{attribute 'linkalways'} 
{attribute 'no_explicit_call' := 'This FB is a CLASS and must be accessed using methods or properties'}
{attribute 'enable_dynamic_creation'}
FUNCTION_BLOCK Node_F_VN_ConvexHullPointsExp EXTENDS VisionNode
VAR
    ipPointSet : _ITcVnContainer;
    ipConvexHull : _ITcVnContainer;
    bClockwise : _BOOL(FALSE);
    hrPrev : _HRESULT(S_OK);
	hresult : _HRESULT(S_OK);
END_VAR

METHOD PUBLIC  Clone : I_Node
VAR
	pNode : POINTER TO Node_F_VN_ConvexHullPointsExp;
END_VAR
pNode := __NEW(Node_F_VN_ConvexHullPointsExp);
Clone := pNode^;
END_METHOD

METHOD FB_init : BOOL
VAR_INPUT
	bInitRetains : BOOL; // if TRUE, the retain variables are initialized (warm start / cold start)
	bInCopyCode : BOOL;  // if TRUE, the instance afterwards gets moved into the copy code (online change)
END_VAR
AddInput('ipPointSet', ipPointSet);
AddParameter('bClockwise', bClockwise);
AddInput('hrPrev', hrPrev);
AddOutput('ipConvexHull', ipConvexHull);
AddOutput('hresult',hresult);
END_METHOD

METHOD PROTECTED OnExecute
hresult.Value := F_VN_ConvexHullPointsExp(
	ipPointSet := ipPointSet.Value,
    ipConvexHull := ipConvexHull.Value,
    bClockwise := bClockwise.Value,
	hrPrev:= hrPrev.Value);
END_METHOD

METHOD PUBLIC PreExecutionCheck
VAR_INPUT
	Check : I_PreExecutionChecks;
END_VAR
Check.IsTrue(ipPointSet.IsValid, 'ipPointSet must be a valid container');
Check.IsTrue((ipPointSet.IsType(TC_GLOBAL_CONST_LIST.ContainerType_Vector_TcVnPoint2_DINT) OR
              ipPointSet.IsType(TC_GLOBAL_CONST_LIST.ContainerType_Vector_TcVnPoint2_REAL)),
              'ipPointSet contains incorrect type');
END_METHOD

END_FUNCTION_BLOCK

(* stored: Version 1.1.0.1, ProductVersion 3.1.4026.13
   POU Node_F_VN_ConvexHullPointsExp: Id {c4240ced-d582-0ee6-3857-2851455c205f}, SpecialFunc None
   Folder Constructor: Id {3e43f53e-70c7-01ef-1900-ee7d664f133a}
   Method Clone: Id {a007ea3e-3cb8-02a6-011b-df6285fba147}
   Method FB_init: Id {9c58b6b3-bcf6-060a-1552-1e0f79d1c8e2}
   Method OnExecute: Id {a86fd9b7-54dd-00d8-0bb6-cbcaa6f3a0fa}
   Method PreExecutionCheck: Id {691c4180-dddf-0bfe-1ad4-27e3b8b091f1} *)
